(* PLC project v0.6.04_CycleSemiAuto.project, CODESYS CODESYS V3.5 SP19 Patch 1 *)
(* stored: creationDateTime 2026-07-27T13:44:41.144048, modificationDateTime 2026-07-27T13:44:41.144048 *)

TYPE ST_ChainWinch : STRUCT
  Inputs_100 : ST_Chain_Winch_Inputs;
  Demandes_200 : ST_Chain_Winch_Demandes;
  Safety_300 : ST_Chain_Winch_Safety;
  Control_400 : ST_Chain_Winch_Control;
  Outputs_500 : ST_Chain_Winch_Outputs;
END_STRUCT;
END_TYPE

TYPE ST_Chain_Winch_Control : STRUCT
  Idx401_MotionAllowed : BOOL;  (* 1 = Prêt / Mouvement Autorisé | 0 = Bloqué *)
  Idx402_SpeedStepCalculated : INT;  (* Palier Vitesse Calculé (0, 1, 2, 3, 4) *)
  Idx403_SpeedRamp_Pct : REAL;  (* [%] Consigne Vitesse après Rampe *)
  Idx404_BrakeReleaseAuthorized : BOOL;  (* 1 = Ordre Ouverture Frein | 0 = Ordre Serrage *)
  Idx405_FinalInterlockState : E_WinchFinalInterlockState;  (* 🛡️ État frontière _LD *)
  Idx406_FinalInterlockReason : E_WinchFinalInterlockReason;  (* 🛡️ Cause mémorisée *)
  Idx407_FinalAuthorizedStep : INT;  (* 🪜 Palier réellement autorisé *)
  Idx408_BrakeCommandOpenConfirmed : BOOL;  (* 🔌 Contacteur/bobine, pas frein mécanique *)
  Idx409_BrakeTimeoutElapsed : TIME;  (* ⏱️ Watchdog 500ms écoulé *)
  Idx410_RestartDelayElapsed : TIME;  (* ⏱️ Verrou 900ms écoulé *)
  Idx411_StepDelayElapsed : TIME;  (* ⏱️ Délai palier 1s250 écoulé *)
  Idx412_InTopSlowdownZone : BOOL;  (* 🆕 2026-08-07 : Palier plafonné à 1, approche limite haute *)
  Idx413_InBottomSlowdownZone : BOOL;  (* 🆕 2026-08-07 : Palier plafonné à 1, approche limite basse (câble ou légale) *)
  Idx414_BottomLimitActiveM : REAL;  (* 🆕 2026-08-07 : Limite basse active (m) — câble physique OU légale, la plus restrictive *)
END_STRUCT;
END_TYPE

TYPE ST_Chain_Winch_Demandes : STRUCT
  Idx201_JoyRawPhysical_ANA : INT;  (* [pts] Bruts convertisseur (-2048 à +2048) *)
  Idx202_JoyScaledPhysical_Pct : REAL;  (* [%] Consigne Joystick (-100% à +100%) *)
  Idx203_HmiManualCmd_BtnUp : BOOL;  (* 1 = Appui Bouton Montée IHM | 0 = Relâché *)
  Idx204_HmiManualCmd_BtnDown : BOOL;  (* 1 = Appui Bouton Descente IHM | 0 = Relâché *)
  Idx205_CycleAutoCmd_Pct : REAL;  (* [%] Consigne auto envoyée par le Cycle *)
  Idx206_ModeActive : E_Mode;  (* Mode courant (MANU_N1, AUTO_N1, MAINT_N2...) *)
  Idx207_BypassOperatorComm : BOOL;  (* 0 = Comm Normale OK | 1 = Bypass Réseau Actif ⚠️ *)
  Idx208_ArbitratedSpeed_Pct : REAL;  (* [%] Consigne finale retenue après arbitrage *)
  Idx209_ArbitratedDirection : INT;  (* +1 = Montée | 0 = Neutre | -1 = Descente *)
  Idx210_CoupledUserRequestDirection : INT;  (* +1 = Montée | 0 = Neutre | -1 = Descente *)
  Idx211_CoupledUserRequestActive : BOOL;  (* 1 = demande utilisateur couplée active *)
END_STRUCT;
END_TYPE

TYPE ST_Chain_Winch_Inputs : STRUCT
  Idx101_EncoderRawPos : DINT;  (* [Valeur brutes pts] Codeur connecté *)
  Idx102_CablePos_M : REAL;  (* [mètres] Position calculée du câble *)
  Idx103_ContactorsReleased_DI : BOOL;  (* 1 = OK (Tous contacteurs retombés à l'arrêt) | 0 = Contacteur collé 🔴 *)
  Idx104_BrakeApplied : BOOL;  (* TRUE = frein SERRÉ (NOT BrakeFeedback — IHM garde le sens serré) *)
  Idx105_ThermalOk_DI : BOOL;  (* 1 = Température OK (Sain) | 0 = Surchauffe Moteur M1 🔴 *)
END_STRUCT;
END_TYPE

TYPE ST_Chain_Winch_Outputs : STRUCT
  Idx501_CmdRelayFwd_Up_DQ : BOOL;  (* 1 = Relais Montée ON | 0 = OFF *)
  Idx502_CmdRelayRev_Down_DQ : BOOL;  (* 1 = Relais Descente ON | 0 = OFF *)
  Idx503_CmdSpeedContactor1_DQ : BOOL;  (* 1 = Contacteur Vitesse 1 ON | 0 = OFF *)
  Idx504_CmdSpeedContactor4_DQ : BOOL;  (* 1 = Contacteur Vitesse 4 ON (Plein Gaz) | 0 = OFF *)
  Idx505_CmdBrakeRelease_RQ : BOOL;  (* 1 = Bobine Frein Alimentée (Ouvert) | 0 = Non Alimentée (Serré) *)
END_STRUCT;
END_TYPE

TYPE ST_Chain_Winch_Safety : STRUCT
  Idx301_EmergencyChainClosed : BOOL;  (* 1 = Boucle Urgence OK (Armé) | 0 = Arrêt d'Urgence Appuyé 🔴 *)
  Idx302_SafeStopActive : BOOL;  (* 0 = Sain (Autorisé) | 1 = Arrêt Rapide Métier Actif 🔴 *)
  Idx303_PowerCutOffActive : BOOL;  (* 0 = Puissance OK | 1 = Coupure Puissance Sécurité 🔴 *)
  Idx304_TopSensorPhysical_DI : BOOL;  (* 1 = Capteur Haut Libre (Sain) | 0 = Butée Haute Atteinte 🔴 *)
  Idx305_TopSensorBypassActive : BOOL;  (* 0 = Capteur Actif | 1 = Capteur Haut Shunté IHM ⚠️ *)
  Idx306_AscentPermitEffective : BOOL;  (* 1 = Montée Autorisée | 0 = MONTÉE BLOQUÉE 🔴 *)
  Idx307_SlackCablePhysical_DI : BOOL;  (* 1 = Câble Tendu (Sain) | 0 = Mou de Câble Détecté 🔴 *)
  Idx308_SlackCableBypassActive : BOOL;  (* 0 = Capteur Actif | 1 = Mou de Câble Shunté IHM ⚠️ *)
  Idx309_DescendPermitEffective : BOOL;  (* 1 = Descente Autorisée | 0 = DESCENTE BLOQUÉE 🔴 *)
  Idx310_MecaFaultMask : WORD;  (* 0 = Pas de Défaut | >0 = Bitfield Défauts Méca A-E 🔴 *)
END_STRUCT;
END_TYPE

{attribute 'qualified_only'}
{attribute 'strict'}
TYPE E_WinchFinalInterlockReason : (NONE := 0, BRAKE_COMMAND_NOT_CONFIRMED := 1, RESTART_INHIBITED := 2);
END_TYPE

{attribute 'qualified_only'}
{attribute 'strict'}
TYPE E_WinchFinalInterlockState : (DISABLED := 0, READY := 1, WAIT_BRAKE_COMMAND_CONFIRMATION := 2, WAIT_STEP_DELAY := 3, WAIT_RESTART_DELAY := 4, FAULT := 5);
END_TYPE

(* values of E_Mode: DISABLE: Mode Désactivé / Veille de sécurité (sorties bloquées); MAINT_N1: Manuel Niveau 1 : Pilotage unitaire avec toutes sécurités actives; MAINT_N2: Manuel Niveau 2 : Pilotage dégradé (droits étendus + bypasses autorisés); SEMI_AUTO: Mode Semi-Automatique (séquenceur automatique) *)

{attribute 'qualified_only'}
{attribute 'strict'}
TYPE E_Mode : (DISABLE := 0, MAINT_N1 := 1, MAINT_N2 := 2, SEMI_AUTO := 3);
END_TYPE
